// TwinCAT 3 PLC project MainPlcProgram
// ProgramVersion: 3.1.4023.0
// libraries:
//   Tc2_Standard, * (Beckhoff Automation GmbH)
//   Tc2_System, * (Beckhoff Automation GmbH)
//   Tc2_Utilities, * (Beckhoff Automation GmbH)
//   Tc3_Module, * (Beckhoff Automation GmbH)
// project tree:
//   CsvLogger/ByteBuffer/ ByteBuffer.TcPOU, ByteBufferFileWriter.TcPOU (not stored), FileBasedByteBuffer.TcPOU, GVL_ByteBufferConstants.TcGVL (not stored)
//   CsvLogger/ByteBuffer/Interface/ I_Buffer.TcIO
//   CsvLogger/CsvDocument/ CsvByteDocumentWriter.TcPOU
//   CsvLogger/CsvDocument/Interfaces/ I_CsvDocument.TcIO (not stored), I_CsvRecord.TcIO
//   / PlcTask.TcTTO (not stored)
//   POUs/ MAIN.TcPOU
// real-time tasks:
//   TASK PlcTask: cycle T#1ms, priority 20, ADS port 350

// ---- CsvLogger/ByteBuffer/Interface/I_Buffer.TcIO
INTERFACE I_Buffer

METHOD PUBLIC AddBoolToBuffer : BOOL
VAR_IN_OUT
	Field : BOOL;
END_VAR
END_METHOD

METHOD PUBLIC AddCharToBuffer : BOOL
VAR_IN_OUT
	Field : BYTE;
END_VAR
END_METHOD

METHOD PUBLIC AddIntToBuffer : BOOL
VAR_IN_OUT
	Field : INT;
END_VAR
END_METHOD

PROPERTY PUBLIC Address : pointer to byte
GET
END_GET
END_PROPERTY

METHOD PUBLIC AddStringToBuffer : BOOL
VAR_IN_OUT
	stringToWrite : STRING;
END_VAR
END_METHOD

METHOD PUBLIC AddULintToBuffer : BOOL
VAR_IN_OUT
	Field : ULINT;
END_VAR
END_METHOD

PROPERTY PUBLIC Remaining : UDINT
GET
END_GET
END_PROPERTY

METHOD PUBLIC Reset
VAR_INPUT
END_VAR
END_METHOD

PROPERTY PUBLIC Size : udint
GET
END_GET
END_PROPERTY

END_INTERFACE

// ---- CsvLogger/CsvDocument/Interfaces/I_CsvRecord.TcIO
INTERFACE I_CsvRecord

METHOD PUBLIC AddBool : I_CsvRecord;
VAR_IN_OUT
	Field : BOOL;
END_VAR
END_METHOD

METHOD PUBLIC AddBoolLiteral : I_CsvRecord;
VAR_INPUT
	Field : BOOL;
END_VAR
END_METHOD

METHOD PUBLIC AddInt : I_CsvRecord;
VAR_IN_OUT
	Field : INT;
END_VAR
END_METHOD

METHOD PUBLIC AddIntLiteral : I_CsvRecord;
VAR_INPUT
	Field : INT;
END_VAR
END_METHOD

METHOD PUBLIC AddString : I_CsvRecord;
VAR_IN_OUT
	stringToWrite : STRING;
END_VAR
END_METHOD

METHOD PUBLIC AddStringLiteral : I_CsvRecord;
VAR_INPUT
	stringToWrite : STRING;
END_VAR
END_METHOD

METHOD PUBLIC EndRecord : I_CsvDocument;
END_METHOD

END_INTERFACE

// ---- CsvLogger/ByteBuffer/ByteBuffer.TcPOU
FUNCTION_BLOCK ByteBuffer implements I_Buffer
VAR_INPUT
END_VAR
VAR_OUTPUT
END_VAR
VAR
	buffer : POINTER TO BYTE;
	bufferSize : UDINT;
	_size : UDINT;
END_VAR
VAR CONSTANT
	SIZE_OF_INT : UDINT := SIZEOF(INT);
	SIZE_OF_ULINT : UDINT := SIZEOF(ULINT);
	SIZE_OF_CHAR : UDINT := SIZEOF(BYTE);
	SIZE_OF_BOOL : UDINT := SIZEOF(BOOL);	
END_VAR

METHOD PUBLIC AddBoolToBuffer : BOOL
VAR_IN_OUT
	Field : BOOL;
END_VAR
IF Remaining >= SIZE_OF_BOOL THEN
	
	memcpy(GetNextAvailableAddress(),ADR(Field),SIZE_OF_BOOL);
	UpdateUsedBufferSize(SIZE_OF_BOOL);

END_IF
END_METHOD

METHOD PUBLIC AddCharToBuffer : BOOL
VAR_IN_OUT
	Field : BYTE;
END_VAR
IF Remaining >= SIZE_OF_CHAR THEN
	
	memcpy(GetNextAvailableAddress(),ADR(Field),SIZE_OF_CHAR);
	UpdateUsedBufferSize(SIZE_OF_CHAR);

END_IF
END_METHOD

METHOD PUBLIC AddIntToBuffer : BOOL
VAR_IN_OUT
	Field : INT;
END_VAR
IF Remaining >= SIZE_OF_INT THEN
	
	memcpy(GetNextAvailableAddress(),ADR(Field),SIZE_OF_INT);
	UpdateUsedBufferSize(SIZE_OF_INT);

END_IF
END_METHOD

PROPERTY PUBLIC Address : pointer to byte
GET
Address := buffer;
END_GET
END_PROPERTY

METHOD PUBLIC AddStringToBuffer : BOOL
VAR_IN_OUT
	stringToWrite : STRING;
END_VAR
VAR
	sizeInBytes : UDINT;
END_VAR
sizeInBytes := INT_TO_UDINT(len(stringToWrite));

IF Remaining >= sizeInBytes THEN
	
	memcpy(GetNextAvailableAddress(),ADR(stringToWrite),sizeInBytes);
	UpdateUsedBufferSize(sizeInBytes);

END_IF
END_METHOD

METHOD PUBLIC AddULintToBuffer : BOOL
VAR_IN_OUT
	Field : ULINT;
END_VAR
IF Remaining >= SIZE_OF_ULINT THEN
	
	memcpy(GetNextAvailableAddress(),ADR(Field),SIZE_OF_ULINT);
	UpdateUsedBufferSize(SIZE_OF_ULINT);

END_IF
END_METHOD

METHOD FB_init : BOOL
VAR_INPUT
	bInitRetains : BOOL; // if TRUE, the retain variables are initialized (warm start / cold start)
	bInCopyCode : BOOL;  // if TRUE, the instance afterwards gets moved into the copy code (online change)
	Buffer : POINTER TO BYTE;
	BufferSize : UDINT;
END_VAR
THIS^.buffer := Buffer;
THIS^.bufferSize := BufferSize;
END_METHOD

METHOD PRIVATE GetNextAvailableAddress : POINTER TO BYTE
VAR_INPUT
END_VAR
GetNextAvailableAddress := buffer + _size;
END_METHOD

PROPERTY PUBLIC Remaining : UDINT
GET
Remaining := bufferSize - _size;
END_GET
END_PROPERTY

METHOD PUBLIC Reset
VAR_INPUT
END_VAR
memset(buffer,16#00,bufferSize);
_size := 0;
END_METHOD

PROPERTY PUBLIC Size : udint
GET
Size := _size;
END_GET
END_PROPERTY

METHOD PRIVATE UpdateUsedBufferSize : BOOL;
VAR_INPUT
	insertFieldSize : UDINT;
END_VAR
_size := _size + insertFieldSize;
END_METHOD

END_FUNCTION_BLOCK

// ---- CsvLogger/ByteBuffer/FileBasedByteBuffer.TcPOU
FUNCTION_BLOCK FileBasedByteBuffer IMPLEMENTS I_Buffer
VAR
	
	fileName : STRING;
	state: (IDLE, START_WRITING, INITIALISE, CYCLIC_WRITE, CLOSE) := IDLE;
	binaryFileWriter : ByteBufferFileWriter('');
		
	buffer1 : ARRAY [0..GVL_ByteBufferConstants.FILE_WRITE_BUFFER_SIZE] OF BYTE;
	buffer2 : ARRAY [0..GVL_ByteBufferConstants.FILE_WRITE_BUFFER_SIZE] OF BYTE;
	byteBuffer1 : ByteBuffer(ADR(buffer1),SIZEOF(buffer1));
	byteBuffer2 : ByteBuffer(ADR(buffer2),SIZEOF(buffer2));
	
	currentlySavingBuffer : I_Buffer := byteBuffer2;
	standbyBuffer : I_Buffer := byteBuffer2;
	activeBuffer : I_Buffer := byteBuffer1;
	
END_VAR

CASE state OF
		
	IDLE: //
	
	START_WRITING: 
	
		byteBuffer1.Reset();
		byteBuffer2.Reset();
		
		activeBuffer := byteBuffer1;
		standbyBuffer := byteBuffer2;
		currentlySavingBuffer := standbyBuffer;
		
		binaryFileWriter.OpenFile(fileName);
		state := CYCLIC_WRITE;
		
	CYCLIC_WRITE: //
		
	CLOSE: 
	
		IF activeBuffer.Size = 0 AND standbyBuffer.Size = 0 THEN
			IF binaryFileWriter.CloseFile() THEN 
				state := IDLE;
			END_IF
		END_IF
	
END_CASE

binaryFileWriter();

IF binaryFileWriter.WriteComplete THEN
	currentlySavingBuffer.Reset();
END_IF

IF standbyBuffer.Size = 0 THEN
	IF binaryFileWriter.WriteByteBufferToFile(activeBuffer) THEN
		currentlySavingBuffer := activeBuffer;
		activeBuffer := standbyBuffer;
		standbyBuffer := currentlySavingBuffer;
	END_IF
END_IF

METHOD PUBLIC AddBoolToBuffer : BOOL
VAR_IN_OUT
	Field : BOOL;
END_VAR
AddBoolToBuffer := activeBuffer.AddBoolToBuffer(Field);
END_METHOD

METHOD PUBLIC AddCharToBuffer : BOOL
VAR_IN_OUT
	Field : BYTE;
END_VAR
AddCharToBuffer := activeBuffer.AddCharToBuffer(Field);
END_METHOD

METHOD PUBLIC AddIntToBuffer : BOOL
VAR_IN_OUT
	Field : INT;
END_VAR
AddIntToBuffer := activeBuffer.AddIntToBuffer(Field);
END_METHOD

PROPERTY PUBLIC Address : pointer to byte
GET
Address := activeBuffer.Address;
END_GET
END_PROPERTY

METHOD PUBLIC AddStringToBuffer : BOOL
VAR_IN_OUT
	stringToWrite : STRING;
END_VAR
AddStringToBuffer := activeBuffer.AddStringToBuffer(stringToWrite);
END_METHOD

METHOD AddULintToBuffer : BOOL
VAR_IN_OUT
	Field	: ULINT;
END_VAR
AddULintToBuffer := activeBuffer.AddULintToBuffer(Field);
END_METHOD

PROPERTY PUBLIC IsActive : BOOL
GET
IsActive := state = CYCLIC_WRITE;
END_GET
END_PROPERTY

PROPERTY PUBLIC IsStopped : BOOL
GET
IsStopped := state = IDLE;
END_GET
END_PROPERTY

PROPERTY PUBLIC Remaining : UDINT
GET
Remaining := activeBuffer.Remaining;
END_GET
END_PROPERTY

METHOD Reset
VAR_INPUT
END_VAR
activeBuffer.Reset();
END_METHOD

PROPERTY PUBLIC Size : udint
GET
Size := activeBuffer.Size;
END_GET
END_PROPERTY

METHOD PUBLIC Start : BOOL
VAR_INPUT
	fileName : STRING;
END_VAR
IF State = IDLE THEN
	THIS^.fileName := fileName;
	State := START_WRITING;
	Start := TRUE;
END_IF
END_METHOD

METHOD PUBLIC Stop : BOOL
VAR_INPUT
END_VAR
IF State = CYCLIC_WRITE THEN
	State := CLOSE;
	Stop := TRUE;
END_IF
END_METHOD

END_FUNCTION_BLOCK

// ---- CsvLogger/CsvDocument/CsvByteDocumentWriter.TcPOU
FUNCTION_BLOCK CsvByteDocumentWriter IMPLEMENTS I_CsvDocument, I_CsvRecord
VAR
	
	byteBuffer : I_Buffer;
	fieldStyle : (NEW_FIELD,NEXT_FIELD) := NEW_FIELD;
	_useQuotes : BOOL := TRUE;
	_fieldCount : UDINT;
	_recordCount : UDINT;
	_fieldDivider : BYTE := F_ToASC(';');
	_recordEnd : STRING := '$0D$0A';
	quoteMark : BYTE := F_ToASC('"'); 
	
END_VAR

METHOD PUBLIC AddBool : I_CsvRecord;
VAR_IN_OUT
	Field : BOOL;
END_VAR
BeforeAddFieldOperations();
byteBuffer.AddBoolToBuffer(Field);
AfterAddFieldOperations();
AddBool := THIS^;
END_METHOD

METHOD PUBLIC AddBoolLiteral : I_CsvRecord;
VAR_INPUT
	Field : BOOL;
END_VAR
BeforeAddFieldOperations();
byteBuffer.AddBoolToBuffer(Field);
AfterAddFieldOperations();
AddBoolLiteral := THIS^;
END_METHOD

METHOD PROTECTED AddFieldDividerToBuffer
byteBuffer.AddCharToBuffer(_fieldDivider);
END_METHOD

METHOD PUBLIC AddInt : I_CsvRecord;
VAR_IN_OUT
	Field : INT;
END_VAR
BeforeAddFieldOperations();
byteBuffer.AddIntToBuffer(Field);
AfterAddFieldOperations();
AddInt := THIS^;
END_METHOD

METHOD PUBLIC AddIntLiteral : I_CsvRecord;
VAR_INPUT
	Field : INT;
END_VAR
BeforeAddFieldOperations();
byteBuffer.AddIntToBuffer(Field);
AfterAddFieldOperations();
AddIntLiteral := THIS^;
END_METHOD

METHOD PROTECTED AddQuoteToBuffer
byteBuffer.AddCharToBuffer(quoteMark);
END_METHOD

METHOD PROTECTED AddRecordEndCharactersToBuffer
byteBuffer.AddStringToBuffer(_recordEnd);
END_METHOD

METHOD PUBLIC AddString : I_CsvRecord;
VAR_IN_OUT
	stringToWrite : STRING;
END_VAR
BeforeAddFieldOperations();
byteBuffer.AddStringToBuffer(stringToWrite);
AfterAddFieldOperations();
AddString := THIS^;
END_METHOD

METHOD PUBLIC AddStringLiteral : I_CsvRecord;
VAR_INPUT
	stringToWrite : STRING;
END_VAR
BeforeAddFieldOperations();
byteBuffer.AddStringToBuffer(stringToWrite);
AfterAddFieldOperations();
AddStringLiteral := THIS^;
END_METHOD

METHOD AddULint : I_CsvRecord
VAR_IN_OUT
	Field	: ULINT;
END_VAR
BeforeAddFieldOperations();
byteBuffer.AddULintToBuffer(Field);
AfterAddFieldOperations();
AddULint := THIS^;
END_METHOD

METHOD AddULintLiteral : I_CsvRecord
VAR_INPUT
	Field	: ULINT;
END_VAR
BeforeAddFieldOperations();
byteBuffer.AddULintToBuffer(Field);
AfterAddFieldOperations();
AddULintLiteral := THIS^;
END_METHOD

METHOD PROTECTED AfterAddFieldOperations
IF _useQuotes THEN
	AddQuoteToBuffer();
END_IF

fieldStyle := NEXT_FIELD;
_fieldCount := _fieldCount + 1;
END_METHOD

METHOD PROTECTED BeforeAddFieldOperations
IF fieldStyle = NEXT_FIELD THEN
	AddFieldDividerToBuffer();
END_IF

IF _useQuotes THEN
	AddQuoteToBuffer();
END_IF
END_METHOD

METHOD PUBLIC EndRecord : I_CsvDocument;
AddRecordEndCharactersToBuffer();
_recordCount := _recordCount + 1;
EndRecord := THIS^;
END_METHOD

METHOD FB_init : BOOL
VAR_INPUT
	bInitRetains : BOOL; // if TRUE, the retain variables are initialized (warm start / cold start)
	bInCopyCode : BOOL;  // if TRUE, the instance afterwards gets moved into the copy code (online change)
	ByteBuffer : I_Buffer;
END_VAR
THIS^.byteBuffer := ByteBuffer;
END_METHOD

PROPERTY PUBLIC FieldCount : UDINT
GET
FieldCount := _fieldCount;
END_GET
END_PROPERTY

PROPERTY PUBLIC FieldDivider : BYTE
GET
FieldDivider := _fieldDivider;
END_GET
SET
_fieldDivider := FieldDivider;
END_SET
END_PROPERTY

PROPERTY PUBLIC IsFull : BOOL
GET
IsFull := byteBuffer.Remaining = 0;
END_GET
END_PROPERTY

PROPERTY PUBLIC RecordCount : UDINT
GET
RecordCount := _recordCount;
END_GET
END_PROPERTY

METHOD Reset
VAR_INPUT
END_VAR
byteBuffer.Reset();
_recordCount := 0;
_fieldCount := 0;
END_METHOD

METHOD PUBLIC StartRecord : reference to CsvByteDocumentWriter//I_CsvRecordWriter
VAR_INPUT
END_VAR
fieldStyle := NEW_FIELD;
StartRecord ref= this^;
END_METHOD

METHOD PUBLIC UpdateBuffer
VAR_INPUT
	Buffer : POINTER TO BYTE;
	BufferSize : UDINT;
END_VAR
END_METHOD

PROPERTY PUBLIC UseQuotes : BOOL
GET
UseQuotes := _useQuotes;
END_GET
SET
_useQuotes := UseQuotes;
END_SET
END_PROPERTY

END_FUNCTION_BLOCK

// ---- POUs/MAIN.TcPOU
PROGRAM MAIN
VAR

	// application
	fileName : STRING := 'C:\myLog.csv';
	targetLogCount : UDINT := 10000; // how many records will be record in the logging session.
	loggingState: (IDLE, INITIALISE, CREATE_HEADER, CYCLIC_LOG_VALUES, COMPLETE_LOGGING) := IDLE;
	maxiumumBufferUsage : UDINT; // you must check this value to make sure it does not exceed GVL_ByteBufferConstants.FILE_WRITE_BUFFER_SIZE
	
	{attribute 'hidden'}
	fileBasedByteBuffer : FileBasedByteBuffer;
	{attribute 'hidden'}
	csvDocumentWriter : CsvByteDocumentWriter(FileBasedByteBuffer);
	{attribute 'hidden'}
	xfcChannel: INT;

	// example data
	SensorName : STRING := 'Sensor1';
	SerialNumber : INT := 123;
	SensorActive : BOOL;
	SensorValue : ARRAY [0..49] OF INT := [1,2,3,4,5,6,7,8,9,10,11,12,13,14,15,16,17,18,19,20,21,22,23,24,25,26,27,28,29,30,31,32,33,34,35,36,37,38,39,40,41,42,43,44,45,46,47,48,49,50];
	
END_VAR

//  Set logging state to INITIALISE to run the example code. 
// --------------------------------------------------------------------------------------------------------------------------------------

CASE loggingState OF
		
	IDLE: 
		// The code will wait here.  You must manually set the loggingState to INITIALISE using the online write values.
	
	INITIALISE:
	
		maxiumumBufferUsage := 0; // this example tracks the maximum buffer usage.  The default buffer size is 200KB.
		
		// The csv document requires a buffer to save the data to.  
		// Therefore before starting to write csv records we must enable the buffer by calling start, plus the file name. 
		
		IF fileBasedByteBuffer.Start(fileName) THEN
			loggingState := CREATE_HEADER;
		END_IF
		
	CREATE_HEADER: 
		
		// This section creates your header information.
		// The information will be stored as bytes.  This example also shows the conversion of an int to string. 
		csvDocumentWriter
			.StartRecord()
			.AddStringLiteral('Sensor Name')
			.AddString(SensorName)
			.EndRecord();	
		csvDocumentWriter
			.StartRecord()
			.AddStringLiteral('Sensor Serial Number')
			.AddStringLiteral(INT_TO_STRING(SerialNumber))
			.EndRecord();
		csvDocumentWriter
			.StartRecord()
			.AddStringLiteral('Column 1')
			.AddStringLiteral('Column 2')
			.AddStringLiteral('Column 3')
			.AddStringLiteral('Column 4')
			.AddInt(SerialNumber)
			.EndRecord();

		loggingState := CYCLIC_LOG_VALUES;
				
	CYCLIC_LOG_VALUES:
			
		// This is the logging section of the code.  You can either make a single record per cycle, or 
		// record multiples based on the array given by our XFC terminals.  In this example I save 50 XFC values plus a few other details
		// Remember, the data is stored as binary.  Use xxx_TO_STRING converters to provide strings. 
		FOR xfcChannel := 0 TO 49 DO   
				csvDocumentWriter
					.StartRecord()
					.AddBool(SensorActive)
					.AddBoolLiteral(TRUE)
					.AddInt(SensorValue[xfcChannel]) 
					.AddIntLiteral(0)
					.EndRecord();
					
		END_FOR
		
		// This controls how many records are written.  You can either use a timer countdown or a record count.  
		// in this example I check the records created and once I have over 300 (including the header) then I complete.
		IF csvDocumentWriter.RecordCount > targetLogCount THEN
			loggingState := COMPLETE_LOGGING;
		END_IF
		
	COMPLETE_LOGGING: 
		
		// You must stop the file based buffer to close and release the file.  Once the buffer has stopped we can then finish
		// by resetting the csvDocument.  This resets the internal counters.
		fileBasedByteBuffer.Stop();
		
		IF fileBasedByteBuffer.IsStopped THEN
			csvDocumentWriter.Reset();
			loggingState := IDLE;
		END_IF

	
END_CASE

// You must cyclic call this fileBasedByteBuffer to give it procesing time.  There is no requirement to call the csvDocumentWriter as this is 
// all event based. 
fileBasedByteBuffer();

// maxiumumBufferUsage must remain under GVL_ByteBufferConstants.FILE_WRITE_BUFFER_SIZE.  If it exceeds then you will drop values.  In this instance
// make GVL_ByteBufferConstants.FILE_WRITE_BUFFER_SIZE larger. 
IF fileBasedByteBuffer.Size > maxiumumBufferUsage THEN
	maxiumumBufferUsage := fileBasedByteBuffer.Size;
END_IF

END_PROGRAM
